Staubli VAL3: MsgTypeStaubli.dtx

public num READ_IO
public num SET_DRIVE_POWER
public num VELOCITY_CFG
public num VELOCITY_CMD
public num WRITE_SINGLE_IO
